INTERFACE ITF_Component2 EXTENDS ITF_BaseComponent

END_INTERFACE

(* stored: Version 1.1.0.1
   Itf ITF_Component2: Id {024e94b9-1406-089b-2bf3-311cad4657a0} *)
